// TIA Portal V16 export
// export: Created 2022-11-17T15:49:29.3232383Z, ExportSetting WithDefaults, DisplayName Totally Integrated Automation Portal, DisplayVersion V16 Update 6, DisplayName TIA Portal Version Control Interface, DisplayVersion V16 Update 2, DisplayName TIA Portal Openness, DisplayVersion V16 Update 6, DisplayName SINAMICS Startdrive Advanced, DisplayVersion V16 Update 5, DisplayName SINAMICS Startdrive G130, G150, S120, S150, SINAMICS MV, S210, DisplayVersion V16 Update 5, DisplayName SINAMICS Startdrive G110M, G120, G120C, G120D, G120P, G115D, DisplayVersion V16 Update 5, DisplayName STEP 7 Professional, DisplayVersion V16 Update 6, DisplayName STEP 7 Safety, DisplayVersion V16, DisplayName WinCC Advanced, DisplayVersion V16 Update 6
FUNCTION "FC81_Optional" : Void   // FC81, LAD
TITLE = Optional
{ S7_Optimized_Access := 'TRUE' }
VERSION : 0.1
// stored: AutoNumber false, IsIECCheckEnabled false, SetENOAutomatically false, UDAEnableTagReadback false
BEGIN

REGION Network 1: Signal Automatic
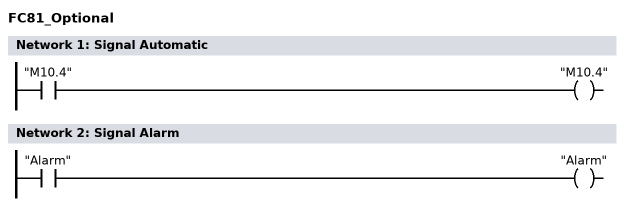
   RUNG wire#powerrail
      Contact( "M10.4" )
      Coil( "M10.4" )
   END_RUNG
   // the same network as SCL:
   "M10.4" := "M10.4";
END_REGION

REGION Network 2: Signal Alarm
   RUNG wire#powerrail
      Contact( "Alarm" )
      Coil( "Alarm" )
   END_RUNG
   // the same network as SCL:
   "Alarm" := "Alarm";
END_REGION
END_FUNCTION
